// Mitsubishi GX Works2 project: test_in_out_blink   PLC: FX3U/FX3UC

PROGRAM MAIN
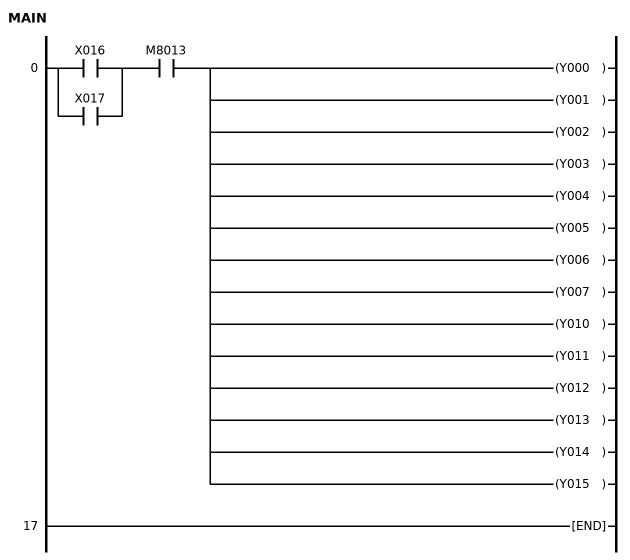
0     LD      X016
      OR      X017
      AND     M8013
      OUT     Y000
      OUT     Y001
      OUT     Y002
      OUT     Y003
      OUT     Y004
      OUT     Y005
      OUT     Y006
      OUT     Y007
      OUT     Y010
      OUT     Y011
      OUT     Y012
      OUT     Y013
      OUT     Y014
      OUT     Y015
17    END
END_PROGRAM
